Staubli VAL3: aLight3.pgx

public program aLight3(num nValue (dimensions=1))
begin
  aioSet(aLight3,nValue)
end
